{attribute 'qualified_only'}
{attribute 'strict'}
TYPE eUpstreamComm : 
(
	indexGroup := eAdsIndexGroups.PLCADS_RWM,
	offsetUpstreamSyncEngaged := 127,
	offsetUpstreamSyncAckowledged := 128
);
END_TYPE

(* stored: Version 1.1.0.1, ProductVersion 3.1.4020.12
   DUT eUpstreamComm: Id {fc112c8e-d256-4f09-ab0d-72667210437a} *)
